FUNCTION_BLOCK FB_Dil_SetValveConfig
VAR_INPUT
	bExecute	: BOOL;
	eValveType  : E_DilValveType;
END_VAR
VAR_OUTPUT
	bBusy		: BOOL;
	bError		: BOOL;
	nErrorId	: ERRORID;
END_VAR
VAR
	nState		: USINT;
	sSendData	: STRING(100);
	timer		: TON;
END_VAR
VAR_IN_OUT
	DilSendCmd 	: FB_Dil_SendCmd;
	pDilRef		: POINTER TO FB_HwRefDiluter;
END_VAR

IF pDilRef = 0 THEN
	bError := TRUE;
	RETURN;	
END_IF

IF bExecute THEN
	CASE nState OF
		0:	//Write valve config
			bBusy := TRUE;
			sSendData := CONCAT(USINT_TO_STRING(pDilRef^.nChannel),'U');
			sSendData := CONCAT(sSendData,USINT_TO_STRING(eValveType));
			sSendData := CONCAT(sSendData,'R');
			DilSendCmd(bExecute:= TRUE, bExpectReply:= TRUE, sSendData:= sSendData);
			
			IF NOT DilSendCmd.bBusy THEN
				IF DilSendCmd.bError THEN
					bBusy := FALSE;
					bError := TRUE;
					nErrorId := DilSendCmd.nErrorId;
				ELSE
					nState := 1;
				END_IF
				DilSendCmd(bExecute:= FALSE);
			END_IF
		
		1:	//Reset
			sSendData := CONCAT(USINT_TO_STRING(pDilRef^.nChannel),'!R');
			DilSendCmd(bExecute:= TRUE, bExpectReply:= FALSE, sSendData:= sSendData);
			IF NOT DilSendCmd.bBusy THEN
				IF DilSendCmd.bError THEN
					bBusy := FALSE;
					bError := TRUE;
					nErrorId := DilSendCmd.nErrorId;
				ELSE
					nState := 2;
				END_IF
				DilSendCmd(bExecute:= FALSE);
			END_IF
		
		2:	//200ms warten, bis Diluter wieder bereit
			timer(IN:= TRUE, PT:=T#200MS);
			IF timer.Q THEN
				timer(IN:= FALSE);
				nState := 80;
				bBusy := FALSE;
			END_IF
	END_CASE
ELSE
	DilSendCmd(bExecute:= FALSE);
	bBusy := FALSE;
	bError := FALSE;
	nErrorId := 0;
	nState := 0;
END_IF

END_FUNCTION_BLOCK

(* stored: Version 1.1.0.1, ProductVersion 3.1.4024.9
   POU FB_Dil_SetValveConfig: Id {264528c4-5071-48be-a466-57fa25d76f4a}, SpecialFunc None *)
